TYPE UNIFIED_PROGRAM_STEP_TRANSITION :
STRUCT
	Condition : UNIFIED_PROGRAM_STEP_TRANSITION_CONDITION;
	Target : BYTE;
END_STRUCT
END_TYPE

(* stored: Version 1.1.0.1
   DUT UNIFIED_PROGRAM_STEP_TRANSITION: Id {834c9ef9-4cff-4ae4-8f34-cf4a19da6d70} *)
